PROGRAM Horizontal_Calibration
VAR
END_VAR

astAxes[AXIS_HORIZONTAL_CALIBRATION].stControl.bEnable := TRUE;
astAxes[AXIS_HORIZONTAL_CALIBRATION].stInputs.bLimitBwd := astAxes[AXIS_HORIZONTAL_TRANSLATION].stInputs.bLimitBwd;
astAxes[AXIS_HORIZONTAL_CALIBRATION].stInputs.bLimitFwd := astAxes[AXIS_HORIZONTAL_TRANSLATION].stInputs.bLimitFwd;

END_PROGRAM

(* stored: Version 1.1.0.1, ProductVersion 3.1.4024.11
   POU Horizontal_Calibration: Id {c5945fad-dfbd-4165-83d8-68115d1e0a8c}, SpecialFunc None *)
